(* PLC project project.ecp, WAGO e!COCKPIT e!COCKPIT *)
(* stored: creationDateTime 2022-06-27T09:59:55.2745601, modificationDateTime 2022-06-27T09:59:23.0778894 *)

TYPE strct : STRUCT
  vari : INT;
END_STRUCT;
END_TYPE

{attribute 'qualified_only'}
{attribute 'strict'}
TYPE enu : (enum_member := 0);
END_TYPE

{attribute 'qualified_only'}
VAR_GLOBAL  (* GVL *)
  myGlobal : INT;
END_VAR

FUNCTION_BLOCK function_blk
  VAR_INPUT
    inVar : INT;
  END_VAR
  VAR
    vari : INT;
  END_VAR
  VAR_OUTPUT
    outVar : INT;
  END_VAR
  VAR_IN_OUT
    inOut : INT;
  END_VAR
  VAR_TEMP
    inOut : INT;
  END_VAR

            
          
END_FUNCTION_BLOCK
